// Registers an I_Execute owner for cyclic execution.
FUNCTION_BLOCK FINAL Execute IMPLEMENTS _I_Execute, I_Debug, I_ValidateInterface
VAR
	_iThread: I_Thread := _Plant.MainThread;
	{attribute 'no_copy'}
	{attribute 'no_init'}
	_iExecute: I_Execute;
	_iPrev: _I_Execute;
	_iNext: _I_Execute;
END_VAR

METHOD INTERNAL _Exe
VAR_OUTPUT
	iNext: _I_Execute;
END_VAR
_iExecute.Execute();
iNext := _iNext;
END_METHOD

METHOD INTERNAL GetNext : _I_Execute
GetNext := _iNext;
END_METHOD

METHOD INTERNAL SetNext
VAR_INPUT
	iNext: _I_Execute;
END_VAR
_iNext := iNext;
END_METHOD

METHOD INTERNAL GetPrev : _I_Execute
GetPrev := _iPrev;
END_METHOD

METHOD INTERNAL SetPrev
VAR_INPUT
	iPrev: _I_Execute;
END_VAR
_iPrev := iPrev;
END_METHOD

METHOD INTERNAL GetThread : I_Thread
GetThread := _iThread;
END_METHOD

METHOD INTERNAL SetThread
VAR_INPUT
	iThread: I_Thread;
END_VAR
_iThread := iThread;
END_METHOD

//FB_Exit must be implemented explicitly. If there is an implementation, then the
//method is called before the controller removes the code of the function block instance
//(implicit call). The return value is not evaluated.
{attribute 'hide'}
METHOD FB_Exit: BOOL
VAR_INPUT
    bInCopyCode: BOOL;  // TRUE: the exit method is called in order to leave the instance which will be copied afterwards (online change).  
END_VAR
IF NOT bInCopyCode THEN
	_iThread.DetachExecute(THIS^);
END_IF
END_METHOD

// Registers iExecute during initialization; panics if iExecute is 0.
{attribute 'hide'}
METHOD FB_Init: BOOL
VAR_INPUT
    bInitRetains: BOOL; // TRUE on retain initialization.
    bInCopyCode: BOOL;  // TRUE before online-change copy.
	
	iExecute			: I_Execute; // Owner to execute cyclically; must not be 0.
END_VAR
IF (_iExecute := iExecute) = 0 THEN
	Plant.Panic(THIS^, Tc2_Standard.CONCAT(__POUNAME(), ': Itf = 0!'));
	RETURN;
END_IF

IF bInCopyCode THEN
	RETURN;
END_IF

_iThread := _Plant.MainThread;
_Plant.MainThread.AttachExecute(THIS^);
END_METHOD

// Thread that runs this executor; set during initialization.
PROPERTY Thread : I_Thread
GET
Thread := _iThread;
END_GET
SET
IF NOT Plant.IsInit THEN
	RETURN;
END_IF

_iThread := Thread;
END_SET
END_PROPERTY

{attribute 'hide'}
METHOD ValidateInterface
END_METHOD

END_FUNCTION_BLOCK

(* stored: Version 1.1.0.1
   POU Execute: Id {fd30bbbf-c4e7-4255-aff2-259a2cee51d5}, SpecialFunc None
   Method _Exe: Id {c801d5e7-2cd0-4874-a9b5-b0187da63b5c}
   Method GetNext: Id {3d96c1fb-39f0-442f-9718-f6d5a86e211b}
   Method SetNext: Id {677f2992-18c1-4c5a-b2ec-d486da3438ff}
   Method GetPrev: Id {3b3ff7c6-bb9b-4733-bc64-54d2c8dcb4cd}
   Method SetPrev: Id {44730286-9026-4f66-98e9-3d355cd1aaea}
   Method GetThread: Id {72227220-0359-407a-8720-7719b42011bf}
   Method SetThread: Id {2857cd8b-9e67-46ff-a686-f2ae4abe909f}
   Method FB_Exit: Id {fbaf27a8-1c97-413f-b76d-2e38666e1e5d}
   Method FB_init: Id {0c4d921f-e0eb-4cc3-851c-9a1e40abf9a1}
   Property Thread: Id {007dbe53-a2a0-4e0f-80d9-08047f4a945c}
   Get Get: Id {b47347c0-efdb-4ac8-ad7a-d8c017d37951}
   Set Set: Id {476d1068-41d5-4d10-b792-0c8db1cb2340}
   Method ValidateInterface: Id {b5b5eaed-d558-4ece-b8e0-6e522161a80d} *)
